FUNCTION_BLOCK MOD_LINT (* IEC 61131-3,Table 24#16 *)
  (* Standard: 61131-3 *)
  (* Version 0.0, 2004-12-15, JHC, Rockwell Automation, Converted from SRC format. *)
  (* Compiler header: package fb.rt.plc.math; *)
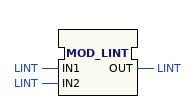
  VAR_INPUT
    IN1 : LINT;
    IN2 : LINT;
  END_VAR
  VAR_OUTPUT
    OUT : LINT;
  END_VAR
END_FUNCTION_BLOCK
